Fanuc KAREL source: kt00124.KL

-- PROVISIONAL review KL for V770-1; original PC SHA256 03374c87f1c066a586f2d5edaae4823ec5d3a9eb237c84597cc2ac958e2646e2
-- Incomplete behavior may be omitted. Consult companion uncertainty JSON. Do not deploy.
PROGRAM KT00124
%NOLOCKGROUP
VAR
  R2 : REAL
  OUT : REAL
-- UNRESOLVED_DECL H1 type=002017
BEGIN
  -- UNRESOLVED_PC offsets 5-19; opcodes 2E,22,9D,33,B4
  -- UNRESOLVED_PC offsets 24-35; opcodes 2E,23
  -- UNRESOLVED_PC offsets 40-65; opcodes 22,9D,33,B3,21,29,64,29,6C,23
  -- UNRESOLVED_PC offsets 70-74; opcodes 7F
END KT00124
